{attribute 'OPC.UA.DA' := '1'}
FUNCTION_BLOCK LightspeedChamber EXTENDS ChamberBase
VAR_INPUT
	IoLightspeed : IoLightspeed;	
	IoSafetyLS : IoSafetyLS;
END_VAR
VAR_OUTPUT
	MppcActivate : BOOL;
END_VAR
VAR
	{attribute 'OPC.UA.DA' := '0'}
	_config : LightspeedChamberConfig;	
	
	{attribute 'OPC.UA.DA' := '0'}
	_initDevice : BOOL;
	
	{attribute 'OPC.UA.DA' := '0'}
	_itemInit : INT;
	{attribute 'OPC.UA.DA' := '0'}
	_pulseGeneratorInit : TON;
	
END_VAR

MppcActivate := IoLightspeed.OutputMppcActivate;

// Init device
InitDevice();

METHOD FB_init : BOOL
VAR_INPUT
	bInitRetains : BOOL; // if TRUE, the retain variables are initialized (warm start / cold start)
	bInCopyCode : BOOL;  // if TRUE, the instance afterwards gets moved into the copy code (online change)
	Config : LightspeedChamberConfig;
END_VAR
IF Config.IsEnabled THEN
	_config := Config;	

	SUPER^._chamberConfig.Name := Config.Name;
	SUPER^._chamberConfig.DeviceID := Config.DeviceID;
	SUPER^._chamberConfig.IsEnabled := Config.IsEnabled;
	SUPER^._chamberConfig.LogLevel := Config.LogLevel;
	
	SUPER^.Name := Config.Name;
	SUPER^.DeviceID := Config.DeviceID;
	
	THIS^.Family := DeviceFamily.Chamber;

	THIS^.SetReady();
	_Logger.Information(_message.Reset().Append('Init ').
							Append('{').Append(TO_STRING(THIS^.Family)).Append('} - ').
							Append('{').Append(TO_STRING(THIS^.Name)).Append('} - ').
							Append('Status : ').Append(TO_STRING(THIS^.Status)).
							ToString());										 
END_IF
END_METHOD

METHOD InitDevice
VAR_INPUT
END_VAR
IF NOT _initDevice THEN			
	IF _pulseGeneratorInit.Q THEN
		_pulseGeneratorInit(IN := FALSE, PT := T#10MS);
			
		CASE _itemInit OF
			0:  _itemInit := 1;
				
			1: _logger.Information(_message.Reset().
								Append(_config.Name).
								Append(' - CoolingFans started').ToString());		
								
				IoLightspeed.OutputCoolingFanFrontPanel := TRUE;
				IoLightspeed.OutputCoolingFanBackPanel := TRUE;
				_initDevice := TRUE;
				_itemInit := 0;
		END_CASE
	ELSE
		_pulseGeneratorInit(IN := TRUE, PT := Const.ACTIVE_TIME_COOLING_FAN);	
	END_IF
END_IF
END_METHOD

{attribute 'TcRpcEnable' := '1'}
METHOD MoveSlitDoorPosition
VAR_INPUT
	Execute : BOOL;
	Position : INT;
END_VAR
IF Execute THEN
	_logger.Information(_message.Reset().Append(_config.Name).Append(' - Move slit door position : ').Append(TO_STRING(Position)).ToString());		

END_IF
END_METHOD

METHOD ReadSlitDoorPosition 
VAR_INPUT
END_VAR
VAR
	open : BOOL;
	close : BOOL;
END_VAR
END_METHOD

END_FUNCTION_BLOCK

(* stored: Version 1.1.0.1, ProductVersion 3.1.4024.12
   POU LightspeedChamber: Id {7ff6493c-add0-491a-9f43-8bd5fbf67492}, SpecialFunc None
   Folder Commands: Id {251073a4-7a66-4518-af59-05416b798691}
   Method FB_init: Id {93f57cf8-52ea-4dbb-91f8-5905b0c1e185}
   Method InitDevice: Id {ecd734fe-ccb4-44d0-a69f-af8966f318b1}
   Method MoveSlitDoorPosition: Id {4b857c95-e373-4ecf-9dbb-168ca7b2be4f}
   Method ReadSlitDoorPosition: Id {34ae610f-f04b-409a-b450-c1fc13e31e1b} *)
